FUNCTION SetSuctionsPtr : BOOL
VAR_INPUT
	suctions : POINTER TO SuctionPad;
	numPads : DINT;
	
	state : BOOL;
END_VAR
VAR
	i : DINT;
END_VAR

FOR i:=0 TO numPads-1 BY 1 DO
	suctions[i].enable := state;
END_FOR

END_FUNCTION

(* stored: Version 1.1.0.1, ProductVersion 3.1.4024.11
   POU SetSuctionsPtr: Id {cf159f8a-7751-40dd-80c3-28a36de916ff}, SpecialFunc None *)
